FUNCTION_BLOCK EL4018
VAR
	_io : EL4xx8_Data;
	{attribute addProperty Name "WcState"}
	_wcState : WcStateBase;
	{attribute addProperty Name "Info data"}
	_infoData : InfoDataAds;
END_VAR

PROPERTY IO : REFERENCE TO EL4xx8_Data
GET
IO REF= _io;
END_GET
END_PROPERTY

PROPERTY WcState : REFERENCE TO WcStateBase
GET
WcState REF= _wcState;
END_GET
END_PROPERTY

END_FUNCTION_BLOCK

(* stored: Version 1.1.0.1, ProductVersion 3.1.4024.9
   POU EL4018: Id {b73ae929-a607-0847-3861-68e8e876292b}, SpecialFunc None
   Property IO: Id {ee0b5ae1-5823-0158-1dff-358db5f5cc48}
   Get Get: Id {cb4ddfec-6eea-087f-3941-1905463ba824}
   Property WcState: Id {9ebe1272-0573-0a06-3d8d-75b5d6b0043a}
   Get Get: Id {867f06e3-bd2e-0b85-2627-1e2f8ac04759} *)
